Fanuc TP program (LS listing): mv_home.ls

/PROG  MV_HOME
/ATTR
DEFAULT_GROUP	= 1,*,*,*,*;
/MN
 : UFRAME_NUM=${WORLD} ;
 : UTOOL_NUM=${FACEPLATE} ;
 : J PR{HOME} ${HOME_SPEED}% CNT0 ;
/POS
/END
